Staubli VAL3: make_NUM.pgx

program make_NUM(string& x_sItem)
  local string l_sMessage
  local num i
  local num l_nValue
  local string l_sEmpty
  local string l_sItem
begin
  cls()
  //
  // = =NUM +1 -1
  //
  // display the actual item
  call use:type(2,12,x_sItem)
  // Select the operator
  call language:message(l_sMessage,110)
  call use:questionDialog(l_sMessage,saveInOut:sOperator,i)
  if i!=-1
    // compose the istruction
    call use:type(2,12,x_sItem+saveInOut:sOperator[i-1])
    // modify the value
    if i==1
      // modify the actual item
      call language:message(l_sMessage,111)
      call use:changeValue(l_nValue,-10000,10000,4+len(x_sItem),12,l_sEmpty)
      x_sItem=x_sItem+saveInOut:sOperator[i-1]+toString("",l_nValue)
    elseIf i==2
      // select a new value
      call selectType(l_sItem)
      if l_sItem!=""
        x_sItem=x_sItem+"=NUM "+l_sItem
      else
        x_sItem=""
      endIf
    elseIf i>2
      // use the + - 1
      x_sItem=x_sItem+saveInOut:sOperator[i-1]
    else
      // escape -> return
    endIf
  endIf
  // validate
  if use:bUseEscape
    x_sItem=""
  endIf
end
